// Block: ProductionMng_PERS

DATA_BLOCK ProductionMng_PERS
VERSION : 0.1
   NON_RETAIN
   VAR
      Pers : Prod_Pers;
   END_VAR

BEGIN
   // No initialization required
END_DATA_BLOCK
